FUNCTION_BLOCK TcoDataExchange EXTENDS TcoCore.TcoObject IMPLEMENTS ITcoCrud
VAR
    _createTask : TcoDataTask(THIS^);
    _readTask : TcoDataTask(THIS^);
    _updateTask : TcoDataTask(THIS^);
    _deleteTask : TcoDataTask(THIS^);
	_idExistsTask : TcoExistsTask(THIS^);
	_createOrUpdateTask : TcoDataTask(THIS^);
END_VAR

_createTask();
_readTask();
_updateTask();
_deleteTask();
_idExistsTask();
_createOrUpdateTask();

(*~
	<docu>
		<summary>
			Creates new entry in the Repository. 	
		</summary>			
		<remarks>
		   <note type="information">
				Inxton is required for this feature to work.
		   </note>	
		</remarks>	
		<example>			
			[!code-pas[Main](~/../TcOpen/src/TcoData/src/XAE/XAE/TcoDataTests/POUs/Sandbox/SandboxContext.TcPOU?name=CreateCodeExample)]
		</example>
	</docu>	
~*)
METHOD Create : TcoCore.ITcoTaskStatus
VAR_INPUT
	(*~
	<docu>
		<summary>
			<remarks>Inxton is required for this feature to work</remarks> 	
		</summary>			
				
	</docu>	
	~*)	
	Identifier : STRING(255);
END_VAR
Create := _createTask
    .WithId(Identifier)
    .Invoke();
	
THIS^.Messenger.Build().Append('<#Creating data item with id:#> ').Append(Identifier).As().AsInfo();
END_METHOD

METHOD CreateOrUpdate : TcoCore.ITcoTaskStatus
VAR_INPUT
	Identifier : STRING(255);
END_VAR
CreateOrUpdate := _createOrUpdateTask
    			  .WithId(Identifier)
                  .Invoke();
				  
THIS^.Messenger.Build().Append('<#Creating or updating data item with id:#> ').Append(Identifier).As().AsInfo();
END_METHOD

METHOD Delete : TcoCore.ITcoTaskStatus
VAR_INPUT
	Identifier : STRING(255);
END_VAR
Delete := _deleteTask
    .WithId(Identifier)
    .Invoke();
	
THIS^.Messenger.Build().Append('<#Deleting data item with id:#> ').Append(Identifier).As().AsInfo();
END_METHOD

METHOD Exists : REFERENCE TO  TcoExistsTask
VAR_INPUT
	Identifier : STRING(255);
END_VAR
_idExistsTask
    .WithId(Identifier)
    .Invoke();

THIS^.Messenger.Build().Append('<#Checking existence of data item with id:#> ').Append(Identifier).As().AsInfo();
	
Exists REF=	_idExistsTask;
END_METHOD

METHOD FB_init : BOOL
VAR_INPUT
	bInitRetains : BOOL; // if TRUE, the retain variables are initialized (warm start / cold start)
	bInCopyCode : BOOL;  // if TRUE, the instance afterwards gets moved into the copy code (online change)
	Parent : TcoCore.ITcoObject;
END_VAR
SUPER^.FB_init(bInitRetains := bInitRetains, bInCopyCode := bInCopyCode, Parent := Parent);
END_METHOD

METHOD Read : TcoCore.ITcoTaskStatus
VAR_INPUT
	Identifier : STRING(255);
END_VAR
Read := _readTask
    .WithId(Identifier)
    .Invoke();
	
THIS^.Messenger.Build().Append('<#Reading data item with id:#> ').Append(Identifier).As().AsInfo();
END_METHOD

METHOD Update : TcoCore.ITcoTaskStatus
VAR_INPUT
	Identifier : STRING(255);
END_VAR
Update := _updateTask
    .WithId(Identifier)
    .Invoke();

THIS^.Messenger.Build().Append('<#Updating data item with id:#> ').Append(Identifier).As().AsInfo();
END_METHOD

END_FUNCTION_BLOCK

(* stored: Version 1.1.0.1, ProductVersion 3.1.4024.9
   POU TcoDataExchange: Id {32f44bd8-796a-0ec8-0970-522f256b63cf}, SpecialFunc None
   Method Create: Id {535f62d3-cdf1-09d6-36dd-65bfab4cf00a}
   Method CreateOrUpdate: Id {9e6a9de9-7f41-0de9-0ac9-c27c65910ff9}
   Method Delete: Id {fbf2b4c4-ddcf-0054-1f59-9460c96d51d6}
   Method Exists: Id {027fb448-351a-0f9b-128f-8e14c974683e}
   Method FB_init: Id {320ee7d5-7550-0944-00e6-b2405597b230}
   Method Read: Id {05052219-e02c-06a1-02d0-9241bf3dd3ff}
   Method Update: Id {d5409d9d-f931-0f6c-095c-9c419d838664} *)
